//defines bounds for all HMI inputs
TYPE input_bounds :
STRUCT
	
	linear_speed_low : LREAL := 0.01; //(m/s)
	linear_speed_high: LREAL := 10.0;  //(m/s)

	tension_low : LREAL := 0.5; //(N)
	tension_high : LREAL := 5; //(N)
	
	turn_count_pickup_low : INT := 1;
	turn_count_pickup_high : INT := 1000;
	
	radius_payoff_low : LREAL:=1; //(mm)
	radius_payoff_high : LREAL:=250; //(mm)
	
	radius_pickup_pancake_low : LREAL:=1; //((mm)
	radius_pickup_pancake_high: LREAL:=400; //(mm)
	
	coil_shape_low : INT :=0;
	coil_shape_high : INT :=2;
	
	acceleration_low : LREAL :=0.1; //(m/s)
	acceleration_high : LREAL :=1; //(m/s)
	
	decceleration_low : LREAL :=0.1; //(m^2/s)
	decelleration_high : LREAL :=1; //(m^2/s)

	jerk_low : LREAL:=0.1;
	jerk_high : LREAL:=1;
	
END_STRUCT
END_TYPE

(* stored: Version 1.1.0.1, ProductVersion 3.1.4024.12
   DUT input_bounds: Id {350e6503-6652-40d6-b2eb-f5a82733be9e} *)
